FUNCTION F_SAFETY_StatusFB_TO_TWOHAND : ST_SAFETY_FBTWOHAND
VAR_INPUT
	stFBStatus						: ST_SAFETY_FBStatus; 	(* Struktura ogolna *)
END_VAR

F_SAFETY_StatusFB_TO_TWOHAND.uStatus.stStatusWords	:= stFBStatus;									(* Przepisanie *)
F_SAFETY_StatusFB_TO_TWOHAND.eState 					:= stFBStatus.BState;							(* Ustawienie enum *)
F_SAFETY_StatusFB_TO_TWOHAND.bGeneralError			:= stFBStatus.wDiagnosis <> 0;					(* General Error *)

END_FUNCTION

(* stored: Version 1.1.0.1, ProductVersion 3.1.4022.12
   POU F_SAFETY_StatusFB_TO_TWOHAND: Id {021bffa3-585e-42e4-8133-e71e6848c295}, SpecialFunc None *)
